{attribute addProperty BoxType "EM3701-0000-0016"}
{attribute addProperty Id "AI_InputsAT %I*AI_Inputs_D7666BC23240WcStateAT %I*WcState_F855686C1620InfoDataAT %I*InfoData_BC63D37F80100"}
{attribute addProperty CRC "1799848378"}
{attribute addProperty SizeInBites "128"}
{attribute addProperty SizeInBytes "16"}
TYPE EM3701_F414E23A :
STRUCT
	{attribute addProperty Name "AI_Inputs"}
	AI_Inputs : AI_Inputs_D7666BC2;
	{attribute addProperty Name "WcState"}
	WcState : WcState_F855686C;
	{attribute addProperty Name "InfoData"}
	InfoData : InfoData_BC63D37F;
END_STRUCT
END_TYPE

(* stored: Version 1.2.0.0, ProductVersion 3.1.4024.9
   DUT EM3701_F414E23A: Id {28db3fe3-b1c8-452d-9046-db0f3b6eb77b} *)
